FUNCTION_BLOCK Fb_Truck EXTENDS FB_Vehicle
VAR_INPUT
END_VAR
VAR_OUTPUT
END_VAR
VAR
END_VAR

METHOD VehicleName : STRING
VAR_INPUT
	sName : STRING;
END_VAR
sVehicleName := CONCAT('Truck name is ', sName);
END_METHOD

END_FUNCTION_BLOCK

(* stored: Version 1.1.0.1, ProductVersion 3.1.4024.16
   POU Fb_Truck: Id {9292bc31-f0a9-40d0-badc-f9fec3c645f1}, SpecialFunc None
   Method VehicleName: Id {764ae11f-73c9-45b4-94ab-4cad57498ec1} *)
